// TIA Portal V15.1 export
// export: Created 2024-06-21T08:40:56.2933176Z, ExportSetting WithDefaults, DisplayName Totally Integrated Automation Portal, DisplayVersion V15.1 Update 5, DisplayName TIA Portal Openness, DisplayVersion V15.1 Update 5, DisplayName SINAMICS Startdrive Advanced, DisplayVersion V15.1, DisplayName G130, G150, S120, S150, SINAMICS MV, S210, DisplayVersion V15.1, DisplayName G110M, G120, G120C, G120D, G120P, DisplayVersion V15.1, DisplayName STEP 7 Professional, DisplayVersion V15.1 Update 5, DisplayName STEP 7 Safety, DisplayVersion V15.1, DisplayName WinCC Professional, DisplayVersion V15.1 Update 5, DisplayName SIMATIC Visualization Architect, DisplayVersion V15.1
FUNCTION "LETAFuseModule17_24_CPC20PN-Config" : Void   // FC1408, SCL
{ S7_Optimized_Access := 'TRUE' }
VERSION : 0.1
// stored: AutoNumber false, IsIECCheckEnabled false, SetENOAutomatically False, UDAEnableTagReadback false
   VAR_INPUT
      I_FuseMod17_Used : Bool;   // Fuse module is used
      I_FuseMod17_CH1_NominalCurrent : Int;   // Nominal current for the fuse
      I_FuseMod17_CH1_Name : String;   // Fuse name
      I_FuseMod17_CH1_Description : String;   // Description
      I_FuseMod17_CH2_NominalCurrent : Int;   // Nominal current for the fuse
      I_FuseMod17_CH2_Name : String;   // Fuse name
      I_FuseMod17_CH2_Description : String;   // Description
      I_FuseMod18_Used : Bool;   // Fuse module is used
      I_FuseMod18_CH1_NominalCurrent : Int;   // Nominal current for the fuse
      I_FuseMod18_CH1_Name : String;   // Fuse name
      I_FuseMod18_CH1_Description : String;   // Description
      I_FuseMod18_CH2_NominalCurrent : Int;   // Nominal current for the fuse
      I_FuseMod18_CH2_Name : String;   // Fuse name
      I_FuseMod18_CH2_Description : String;   // Description
      I_FuseMod19_Used : Bool;   // Fuse module is used
      I_FuseMod19_CH1_NominalCurrent : Int;   // Nominal current for the fuse
      I_FuseMod19_CH1_Name : String;   // Fuse name
      I_FuseMod19_CH1_Description : String;   // Description
      I_FuseMod19_CH2_NominalCurrent : Int;   // Nominal current for the fuse
      I_FuseMod19_CH2_Name : String;   // Fuse name
      I_FuseMod19_CH2_Description : String;   // Description
      I_FuseMod20_Used : Bool;   // Fuse module is used
      I_FuseMod20_CH1_NominalCurrent : Int;   // Nominal current for the fuse
      I_FuseMod20_CH1_Name : String;   // Fuse name
      I_FuseMod20_CH1_Description : String;   // Description
      I_FuseMod20_CH2_NominalCurrent : Int;   // Nominal current for the fuse
      I_FuseMod20_CH2_Name : String;   // Fuse name
      I_FuseMod20_CH2_Description : String;   // Description
      I_FuseMod21_Used : Bool;   // Fuse module is used
      I_FuseMod21_CH1_NominalCurrent : Int;   // Nominal current for the fuse
      I_FuseMod21_CH1_Name : String;   // Fuse name
      I_FuseMod21_CH1_Description : String;   // Description
      I_FuseMod21_CH2_NominalCurrent : Int;   // Nominal current for the fuse
      I_FuseMod21_CH2_Name : String;   // Fuse name
      I_FuseMod21_CH2_Description : String;   // Description
      I_FuseMod22_Used : Bool;   // Fuse module is used
      I_FuseMod22_CH1_NominalCurrent : Int;   // Nominal current for the fuse
      I_FuseMod22_CH1_Name : String;   // Fuse name
      I_FuseMod22_CH1_Description : String;   // Description
      I_FuseMod22_CH2_NominalCurrent : Int;   // Nominal current for the fuse
      I_FuseMod22_CH2_Name : String;   // Fuse name
      I_FuseMod22_CH2_Description : String;   // Description
      I_FuseMod23_Used : Bool;   // Fuse module is used
      I_FuseMod23_CH1_NominalCurrent : Int;   // Nominal current for the fuse
      I_FuseMod23_CH1_Name : String;   // Fuse name
      I_FuseMod23_CH1_Description : String;   // Description
      I_FuseMod23_CH2_NominalCurrent : Int;   // Nominal current for the fuse
      I_FuseMod23_CH2_Name : String;   // Fuse name
      I_FuseMod23_CH2_Description : String;   // Description
      I_FuseMod24_Used : Bool;   // Fuse module is used
      I_FuseMod24_CH1_NominalCurrent : Int;   // Nominal current for the fuse
      I_FuseMod24_CH1_Name : String;   // Fuse name
      I_FuseMod24_CH1_Description : String;   // Description
      I_FuseMod24_CH2_NominalCurrent : Int;   // Nominal current for the fuse
      I_FuseMod24_CH2_Name : String;   // Fuse name
      I_FuseMod24_CH2_Description : String;   // Description
   END_VAR
   VAR_IN_OUT
      IO_Config : "ETAFuseCPC20PNConfig";
   END_VAR
BEGIN
   #IO_Config.Fuse[33].Used := #I_FuseMod17_Used;
   #IO_Config.Fuse[33].NominalCurrent := #I_FuseMod17_CH1_NominalCurrent;
   #IO_Config.Fuse[33].Name := #I_FuseMod17_CH1_Name;
   #IO_Config.Fuse[33].Description := #I_FuseMod17_CH1_Description;

   #IO_Config.Fuse[34].Used := #I_FuseMod17_Used;
   #IO_Config.Fuse[34].NominalCurrent := #I_FuseMod17_CH2_NominalCurrent;
   #IO_Config.Fuse[34].Name := #I_FuseMod17_CH2_Name;
   #IO_Config.Fuse[34].Description := #I_FuseMod17_CH2_Description;

   #IO_Config.Fuse[35].Used := #I_FuseMod18_Used;
   #IO_Config.Fuse[35].NominalCurrent := #I_FuseMod18_CH1_NominalCurrent;
   #IO_Config.Fuse[35].Name := #I_FuseMod18_CH1_Name;
   #IO_Config.Fuse[35].Description := #I_FuseMod18_CH1_Description;

   #IO_Config.Fuse[36].Used := #I_FuseMod18_Used;
   #IO_Config.Fuse[36].NominalCurrent := #I_FuseMod18_CH2_NominalCurrent;
   #IO_Config.Fuse[36].Name := #I_FuseMod18_CH2_Name;
   #IO_Config.Fuse[36].Description := #I_FuseMod18_CH2_Description;

   #IO_Config.Fuse[37].Used := #I_FuseMod19_Used;
   #IO_Config.Fuse[37].NominalCurrent := #I_FuseMod19_CH1_NominalCurrent;
   #IO_Config.Fuse[37].Name := #I_FuseMod19_CH1_Name;
   #IO_Config.Fuse[37].Description := #I_FuseMod19_CH1_Description;

   #IO_Config.Fuse[38].Used := #I_FuseMod19_Used;
   #IO_Config.Fuse[38].NominalCurrent := #I_FuseMod19_CH2_NominalCurrent;
   #IO_Config.Fuse[38].Name := #I_FuseMod19_CH2_Name;
   #IO_Config.Fuse[38].Description := #I_FuseMod19_CH2_Description;

   #IO_Config.Fuse[39].Used := #I_FuseMod20_Used;
   #IO_Config.Fuse[39].NominalCurrent := #I_FuseMod20_CH1_NominalCurrent;
   #IO_Config.Fuse[39].Name := #I_FuseMod20_CH1_Name;
   #IO_Config.Fuse[39].Description := #I_FuseMod20_CH1_Description;

   #IO_Config.Fuse[40].Used := #I_FuseMod20_Used;
   #IO_Config.Fuse[40].NominalCurrent := #I_FuseMod20_CH2_NominalCurrent;
   #IO_Config.Fuse[40].Name := #I_FuseMod20_CH2_Name;
   #IO_Config.Fuse[40].Description := #I_FuseMod20_CH2_Description;

   #IO_Config.Fuse[41].Used := #I_FuseMod21_Used;
   #IO_Config.Fuse[41].NominalCurrent := #I_FuseMod21_CH1_NominalCurrent;
   #IO_Config.Fuse[41].Name := #I_FuseMod21_CH1_Name;
   #IO_Config.Fuse[41].Description := #I_FuseMod21_CH1_Description;

   #IO_Config.Fuse[42].Used := #I_FuseMod21_Used;
   #IO_Config.Fuse[42].NominalCurrent := #I_FuseMod21_CH2_NominalCurrent;
   #IO_Config.Fuse[42].Name := #I_FuseMod21_CH2_Name;
   #IO_Config.Fuse[42].Description := #I_FuseMod21_CH2_Description;

   #IO_Config.Fuse[43].Used := #I_FuseMod22_Used;
   #IO_Config.Fuse[43].NominalCurrent := #I_FuseMod22_CH1_NominalCurrent;
   #IO_Config.Fuse[43].Name := #I_FuseMod22_CH1_Name;
   #IO_Config.Fuse[43].Description := #I_FuseMod22_CH1_Description;

   #IO_Config.Fuse[44].Used := #I_FuseMod22_Used;
   #IO_Config.Fuse[44].NominalCurrent := #I_FuseMod22_CH2_NominalCurrent;
   #IO_Config.Fuse[44].Name := #I_FuseMod22_CH2_Name;
   #IO_Config.Fuse[44].Description := #I_FuseMod22_CH2_Description;

   #IO_Config.Fuse[45].Used := #I_FuseMod23_Used;
   #IO_Config.Fuse[45].NominalCurrent := #I_FuseMod23_CH1_NominalCurrent;
   #IO_Config.Fuse[45].Name := #I_FuseMod23_CH1_Name;
   #IO_Config.Fuse[45].Description := #I_FuseMod23_CH1_Description;

   #IO_Config.Fuse[46].Used := #I_FuseMod23_Used;
   #IO_Config.Fuse[46].NominalCurrent := #I_FuseMod23_CH2_NominalCurrent;
   #IO_Config.Fuse[46].Name := #I_FuseMod23_CH2_Name;
   #IO_Config.Fuse[46].Description := #I_FuseMod23_CH2_Description;

   #IO_Config.Fuse[47].Used := #I_FuseMod24_Used;
   #IO_Config.Fuse[47].NominalCurrent := #I_FuseMod24_CH1_NominalCurrent;
   #IO_Config.Fuse[47].Name := #I_FuseMod24_CH1_Name;
   #IO_Config.Fuse[47].Description := #I_FuseMod24_CH1_Description;

   #IO_Config.Fuse[48].Used := #I_FuseMod24_Used;
   #IO_Config.Fuse[48].NominalCurrent := #I_FuseMod24_CH2_NominalCurrent;
   #IO_Config.Fuse[48].Name := #I_FuseMod24_CH2_Name;
   #IO_Config.Fuse[48].Description := #I_FuseMod24_CH2_Description;
END_FUNCTION
